# EPICS autosave request: ioc/AutoSaveRestore/ramp1Menu.req
file configMenu.req P=$(PREFIX), R=$(SUFFIX), CONFIG=$(CONFIG)
file rampSetting.req P=$(PREFIX), R=$(SUFFIX)
